// TIA Portal project "Ventilacion_analoga" (V15)

(* hardware
DEVICE "S7-1200 station_1"  S7-1200 Station
   slot 0: "Rack_0"  S7-1200 Rack  Rack  V1.0
   slot 1: "PLC_1"  CPU 1214C DC/DC/DC  6ES7 214-1AG40-0XB0  V4.2
   slot 2: "AI 4x13BIT_1"  SM 1231 AI4  6ES7 231-4HD30-0XB0  V1.0
   slot 3: "AQ 1x12BIT_1"  AQ1 signal board  6ES7 232-4HA30-0XB0  V1.0
*)

// ===== PLC "PLC_1"  CPU 1214C DC/DC/DC =====

VAR_GLOBAL   // PLC tag table "Tabla de variables estándar"
   "Clock_Byte" AT %MB0 : Byte;
   "Clock_10Hz" AT %M0.0 : Bool;
   "Clock_5Hz" AT %M0.1 : Bool;
   "Clock_2.5Hz" AT %M0.2 : Bool;
   "Clock_2Hz" AT %M0.3 : Bool;
   "Clock_1.25Hz" AT %M0.4 : Bool;
   "Clock_1Hz" AT %M0.5 : Bool;
   "Clock_0.625Hz" AT %M0.6 : Bool;
   "Clock_0.5Hz" AT %M0.7 : Bool;
   "Entrada TC" AT %IW64 : Int;
   "Normalizada TC 0 a 1" AT %MD10 : Real;
   "Temperatura" AT %MD14 : Real;
   "EFC" AT %MD18 : Real;
   "Normalizada EFC 0 a 1" AT %MD22 : Real;
   "Tag_4" AT %QW80 : Int;
   "Inicio" AT %I0.0 : Bool;
   "Paro" AT %I0.1 : Bool;
   "Sis_habilitado" AT %M5.0 : Bool;
   "Tres_ventiladores" AT %M5.1 : Bool;
   "Dos_Veniladores" AT %M5.2 : Bool;
   "Un_Ventilador" AT %M5.3 : Bool;
   "V1" AT %Q0.0 : Bool;
   "V2" AT %Q0.1 : Bool;
   "V3" AT %Q0.2 : Bool;
   "Alarma" AT %Q0.3 : Bool;
   "Reloj" AT %M5.4 : Bool;
END_VAR

// folder: System blocks/Program resources

DATA_BLOCK "T1"   // DB1
{ S7_Optimized_Access := 'TRUE' }
AUTHOR : Simatic
FAMILY : IEC
NAME : IEC_TMR
VERSION : 1.0
// stored: InstanceOfName IEC_TIMER
"IEC_TIMER"
BEGIN
END_DATA_BLOCK

DATA_BLOCK "T2"   // DB2
{ S7_Optimized_Access := 'TRUE' }
AUTHOR : Simatic
FAMILY : IEC
NAME : IEC_TMR
VERSION : 1.0
// stored: InstanceOfName IEC_TIMER
"IEC_TIMER"
BEGIN
END_DATA_BLOCK

// folder: (top level)

FUNCTION "Acondicionamiento" : Void   // FC1, LAD
{ S7_Optimized_Access := 'TRUE' }
VERSION : 0.1
BEGIN

REGION Network 1
   // Acondicionar temperatura de 0 a 150
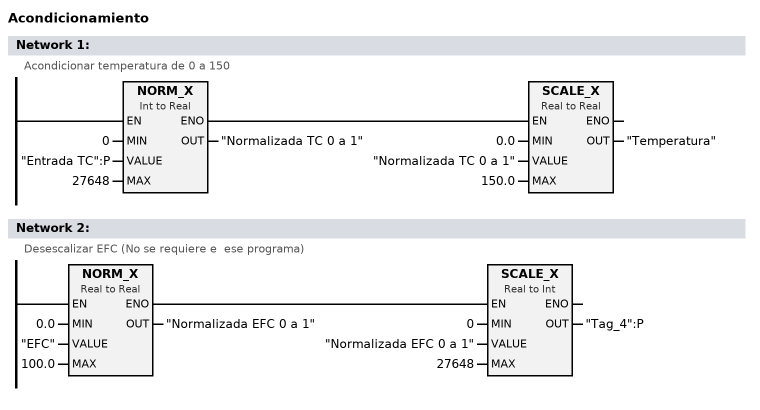
   RUNG wire#powerrail
      { S7_Templates := "[SrcType := Int, DestType := Real]" } Normalize(min := 0, value := "Entrada TC":P, max := 27648, out => "Normalizada TC 0 a 1")
      { S7_Templates := "[SrcType := Real, DestType := Real]" } Scale(min := 0.0, value := "Normalizada TC 0 a 1", max := 150.0, out => "Temperatura")
   END_RUNG
   // the same network as SCL:
   "Normalizada TC 0 a 1" := NORM_X(MIN := 0, VALUE := "Entrada TC":P, MAX := 27648);
   "Temperatura" := SCALE_X(MIN := 0.0, VALUE := "Normalizada TC 0 a 1", MAX := 150.0);
END_REGION

REGION Network 2
   // Desescalizar EFC (No se requiere e  ese programa)
   RUNG wire#powerrail
      { S7_Templates := "[SrcType := Real, DestType := Real]" } Normalize(min := 0.0, value := "EFC", max := 100.0, out => "Normalizada EFC 0 a 1")
      { S7_Templates := "[SrcType := Real, DestType := Int]" } Scale(min := 0, value := "Normalizada EFC 0 a 1", max := 27648, out => "Tag_4":P)
   END_RUNG
   // the same network as SCL:
   "Normalizada EFC 0 a 1" := NORM_X(MIN := 0.0, VALUE := "EFC", MAX := 100.0);
   "Tag_4":P := SCALE_X(MIN := 0, VALUE := "Normalizada EFC 0 a 1", MAX := 27648);
END_REGION
END_FUNCTION

FUNCTION "Control" : Void   // FC2, LAD
{ S7_Optimized_Access := 'TRUE' }
VERSION : 0.1
BEGIN

REGION Network 1
   // Activar el sistema
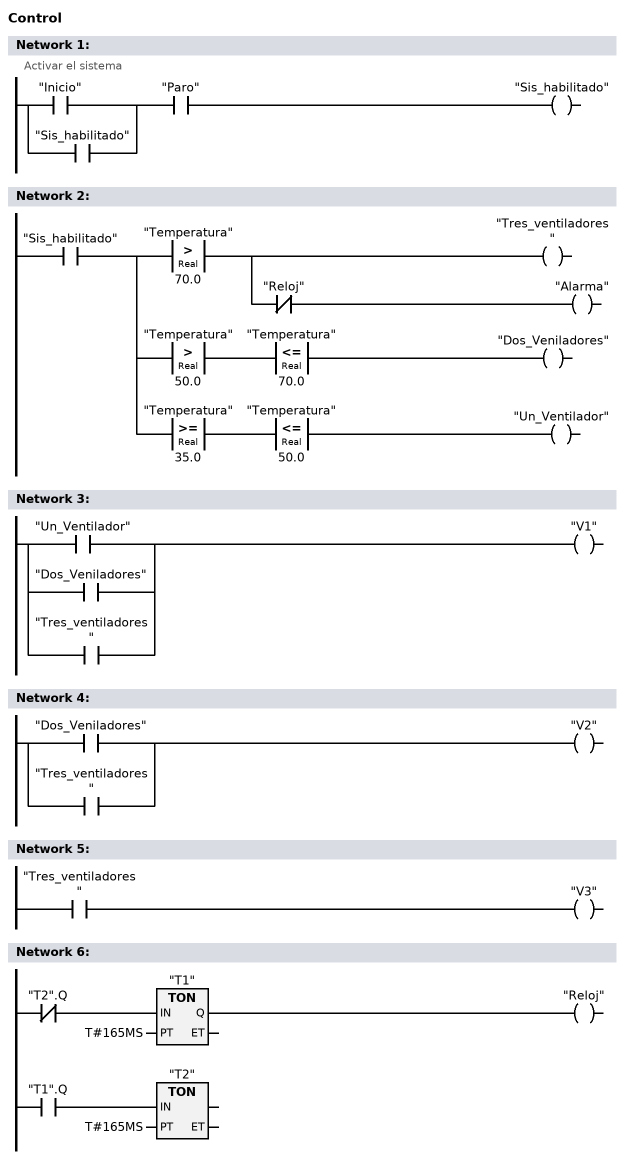
   RUNG wire#powerrail
      Contact( "Inicio" )
      wire#w1
      Contact( "Paro" )
      Coil( "Sis_habilitado" )
   END_RUNG
   RUNG wire#powerrail
      Contact( "Sis_habilitado" )
   END_RUNG wire#w1
   // the same network as SCL:
   "Sis_habilitado" := ("Inicio" OR "Sis_habilitado") AND "Paro";
END_REGION

REGION Network 2
   RUNG wire#powerrail
      Contact( "Sis_habilitado" )
      wire#w1
      { S7_Templates := "SrcType := Real" } GT_Contact(in1 := "Temperatura", in2 := 70.0)
      wire#w2
      Coil( "Tres_ventiladores" )
   END_RUNG
   RUNG wire#w2
      I_Contact( "Reloj" )
      Coil( "Alarma" )
   END_RUNG
   RUNG wire#w1
      { S7_Templates := "SrcType := Real" } GT_Contact(in1 := "Temperatura", in2 := 50.0)
      { S7_Templates := "SrcType := Real" } LE_Contact(in1 := "Temperatura", in2 := 70.0)
      Coil( "Dos_Veniladores" )
   END_RUNG
   RUNG wire#w1
      { S7_Templates := "SrcType := Real" } GE_Contact(in1 := "Temperatura", in2 := 35.0)
      { S7_Templates := "SrcType := Real" } LE_Contact(in1 := "Temperatura", in2 := 50.0)
      Coil( "Un_Ventilador" )
   END_RUNG
   // the same network as SCL:
   "Tres_ventiladores" := "Sis_habilitado" AND ("Temperatura" > 70.0);
   "Alarma" := "Tres_ventiladores" AND NOT "Reloj";
   "Dos_Veniladores" := "Sis_habilitado" AND ("Temperatura" > 50.0) AND ("Temperatura" <= 70.0);
   "Un_Ventilador" := "Sis_habilitado" AND ("Temperatura" >= 35.0) AND ("Temperatura" <= 50.0);
END_REGION

REGION Network 3
   RUNG wire#powerrail
      Contact( "Un_Ventilador" )
      wire#w1
      Coil( "V1" )
   END_RUNG
   RUNG wire#powerrail
      Contact( "Dos_Veniladores" )
   END_RUNG wire#w1
   RUNG wire#powerrail
      Contact( "Tres_ventiladores" )
   END_RUNG wire#w1
   // the same network as SCL:
   "V1" := "Un_Ventilador" OR "Dos_Veniladores" OR "Tres_ventiladores";
END_REGION

REGION Network 4
   RUNG wire#powerrail
      Contact( "Dos_Veniladores" )
      wire#w1
      Coil( "V2" )
   END_RUNG
   RUNG wire#powerrail
      Contact( "Tres_ventiladores" )
   END_RUNG wire#w1
   // the same network as SCL:
   "V2" := "Dos_Veniladores" OR "Tres_ventiladores";
END_REGION

REGION Network 5
   RUNG wire#powerrail
      Contact( "Tres_ventiladores" )
      Coil( "V3" )
   END_RUNG
   // the same network as SCL:
   "V3" := "Tres_ventiladores";
END_REGION

REGION Network 6
   "T1".TON(IN := NOT "T2".Q, PT := T#165MS);
   "Reloj" := "T1".Q;
   "T2".TON(IN := "T1".Q, PT := T#165MS);
END_REGION
END_FUNCTION

ORGANIZATION_BLOCK "Main"   // OB1, LAD, ProgramCycle
TITLE = "Main Program Sweep (Cycle)"
{ S7_Optimized_Access := 'TRUE' }
VERSION : 0.1
   VAR_INPUT
      Initial_Call : Bool;   // Initial call of this OB
      Remanence : Bool;   // =True, if remanent data are available
   END_VAR
BEGIN

REGION Network 1
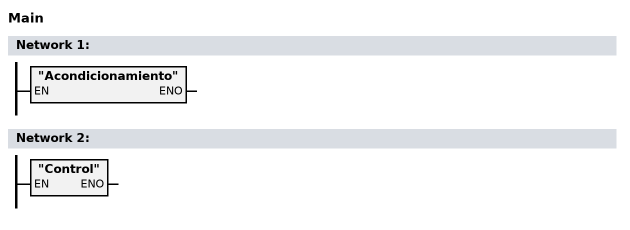
   RUNG wire#powerrail
      "Acondicionamiento"()
   END_RUNG
   // the same network as SCL:
   "Acondicionamiento"();
END_REGION

REGION Network 2
   RUNG wire#powerrail
      "Control"()
   END_RUNG
   // the same network as SCL:
   "Control"();
END_REGION
END_ORGANIZATION_BLOCK